// TIA Portal V18 export
TYPE "PLCtoMES_AGVExchange"
// stored: IsFailsafeCompliant false
   STRUCT
      "P-MaterielCall" : Byte;   // PLC触发物料呼叫信号
      "P-PosCall1" : Byte;   // AGV站点1呼叫（PLC） 1-叫料 2-返空箱 3-空满置换 设备置复位
      "P-PosCall2" : Byte;   // AGV站点2呼叫（PLC） 1-叫料 2-返空箱 3-空满置换 设备置复位
      "P-PosCall3" : Byte;   // AGV站点3呼叫（PLC） 1-叫料 2-返空箱 3-空满置换 设备置复位
      "P-PosCall4" : Byte;   // AGV站点4呼叫（PLC） 1-叫料 2-返空箱 4-空满置换 设备置复位
      "P-PosCall5" : Byte;   // AGV站点5呼叫（PLC） 1-叫料 2-返空箱 4-空满置换 设备置复位
      "P-PalletNo1" : String[38];   // AGV空托盘编号1 38位长度 设备置复位
      "P-PalletNo2" : String[38];   // AGV空托盘编号2 38位长度 设备置复位
      "P-PalletNo3" : String[38];   // AGV空托盘编号3 38位长度 设备置复位
      "P-PalletNo4" : String[38];   // AGV空托盘编号4 38位长度 设备置复位
      "P-PalletNo5" : String[38];   // AGV空托盘编号5 38位长度 设备置复位
      Reserve : Array[1..794] of Byte;   // AGV交互预留
   END_STRUCT;
END_TYPE
